
FUNCTION CB_int_to_word : WORD

TITLE = ' Convert an integer into a word '
VERSION : '1.0'
AUTHOR  : CB
NAME    : intToWor
FAMILY  : TNI

VAR_INPUT
    IN : INT;
END_VAR

BEGIN

CB_int_to_word := INT_TO_WORD(IN);

END_FUNCTION
